(*
    This function resets all test suites that have been initialized.
*)
FUNCTION RERUN_RESET

GVL_TcUnit.TcUnitRunner.ResetTcUnitRunner();

END_FUNCTION

(* stored: Version 1.1.0.1, ProductVersion 3.1.4024.11
   POU RERUN_RESET: Id {5dc2831b-033e-4286-8fb6-238cd06ec5b3}, SpecialFunc None *)
